Yaskawa INFORM job: CUBE_INT_EX.JBI

/JOB
//NAME CUBE_INT_EX
//POS
///NPOS 0,0,0,0,0,0
//INST
///DATE 2016/07/26 17:38
///ATTR SC,RW
NOP
'INTERFERENCE 11 / S2C0013
'CONTROL GROUP: R1 + COMMAND / 65
SET D000 65
SETPRM KIND=5 PRMNO=13 D000
'REF COORDINATE / S2C0087
'0=PULSE 1=BASE 2=ROBOT 3=USER
SET D000 1
SETPRM KIND=5 PRMNO=87 D000
'MAX POSITIONS / S3C0224-S3C0226
'CUBE1 1st POSITION (+) X
SET D000 10000
'CUBE1 1st POSITION (+) Y
SET D001 10000
'CUBE1 1st POSITION (+) Z
SET D002 10000
SETPRM KIND=6 PRMNO=224 D000
SETPRM KIND=6 PRMNO=225 D001
SETPRM KIND=6 PRMNO=226 D002
'MIN POSITIONS / S3C0232-S3C0234
'CUBE1 2nd POSITION (-) X
SET D000 -10000
'CUBE1 2nd POSITION (-) Y
SET D001 -10000
'CUBE1 2nd POSITION (-) Z
SET D002 -10000
SETPRM KIND=6 PRMNO=232 D000
SETPRM KIND=6 PRMNO=233 D001
SETPRM KIND=6 PRMNO=234 D002
END
